TYPE Pos :
STRUCT
	x : REAL;
	y : REAL;
END_STRUCT
END_TYPE

(* stored: Version 1.1.0.1, ProductVersion 3.1.4024.9
   DUT Pos: Id {99a14e6b-1470-4c19-b323-981627db0ea1} *)
